(* Schneider Machine Expert - Basic project ProyekAkhir_Izzudin Al Ayyubi_2006574780, file version 2.7.0.0 *)
(* ProjectInformations: Name=New project *)

HARDWARE
  Cpu 0: TM221CE16R
  EthernetConfiguration: NetworkName=M221, IpAllocationMode=FixedAddress, IpAddress=0.0.0.0, SubnetMask=0.0.0.0
  SerialLineConfiguration: Baud=Baud19200, Parity=ParityEven, DataBits=DataBits8, StopBits=StopBits1, PhysicalMedium=PhysicalMediumRs485, TransmissionMode=TransmissionModeModbusRtu, SlaveId=1, Addressing=SlaveAddressing
  MastTask: UsePeriodScanMode=false, PeriodScan=100
  FastTask: Period=255
  CpuBehavior: StartingMode=StartAsPreviousState, AutoSaveRamOnEeprom=true, WatchdogPeriod=250

SYMBOLS  (address, symbol, comment, settings)
  %M0       MOVING_X
  %M2       ITEM_DETECTED
  %M3       LID_AT_PLACE
  %M4       LID_CLAMPED
  %M6       BASE_AT_PLACE
  %M7       BASE_CLAMPED
  %M9       PARTLEAVING
  %M10      START_
  %M11      RESET
  %M12      STOP
  %M13      EMERGENCYS
  %M14      AUTO
  %M16      MACHINE_BUSY
  %M17      RSENSOR1
  %M18      RSENSOR2
  %M19      VS1_1
  %M20      VS1_2
  %M21      VS2_0
  %M22      VS2_1
  %M23      VS2_3
  %M24      MOVE_X
  %M25      MOVE_Z
  %M26      GRAB
  %M27      LIDSCONVEYOR
  %M28      CLAMP_LID
  %M30      BASECONVEYOR
  %M31      CLAMP_BASE
  %M32      POS_RAISE_BASE
  %M33      STARTLIGHT
  %M34      RESETLIGHT
  %M35      STOPLIGHT
  %M36      MACHINE_START
  %M37      MACHINE_STOP
  %M38      MACHINE_RESET
  %M39      CONVEYOR_MC1
  %M40      CONVEYOR_MC2
  %M41      PIVOT_TURN2
  %M42      PIVOT_TURN3
  %M43      PIVOT_BELT2
  %M44      PIVOT_BELT3
  %M45      PRODUCE_LIDS
  %M46      EMITTER
  %M47      BLUELIGHT
  %M100     STARTMEMORY
  %M101     MEMORY2
  %MW0      COUNTER
  %MW1      DIGITALCOUNTER
  %MW2      VSENSOR1
  %MW3      VSENSOR3
  %TM0        [Preset=1, Base=OneSecond]
  %TM1        [Preset=8, Base=OneHundredMilliSeconds]
  %TM2        [Preset=8, Base=OneHundredMilliSeconds]
  %TM3        [Preset=4, Base=OneHundredMilliSeconds]
  %TM4        [Type=TP, Preset=1500, Base=OneHundredMilliSeconds]

POU New POU
  (* SectionNumber=1 *)

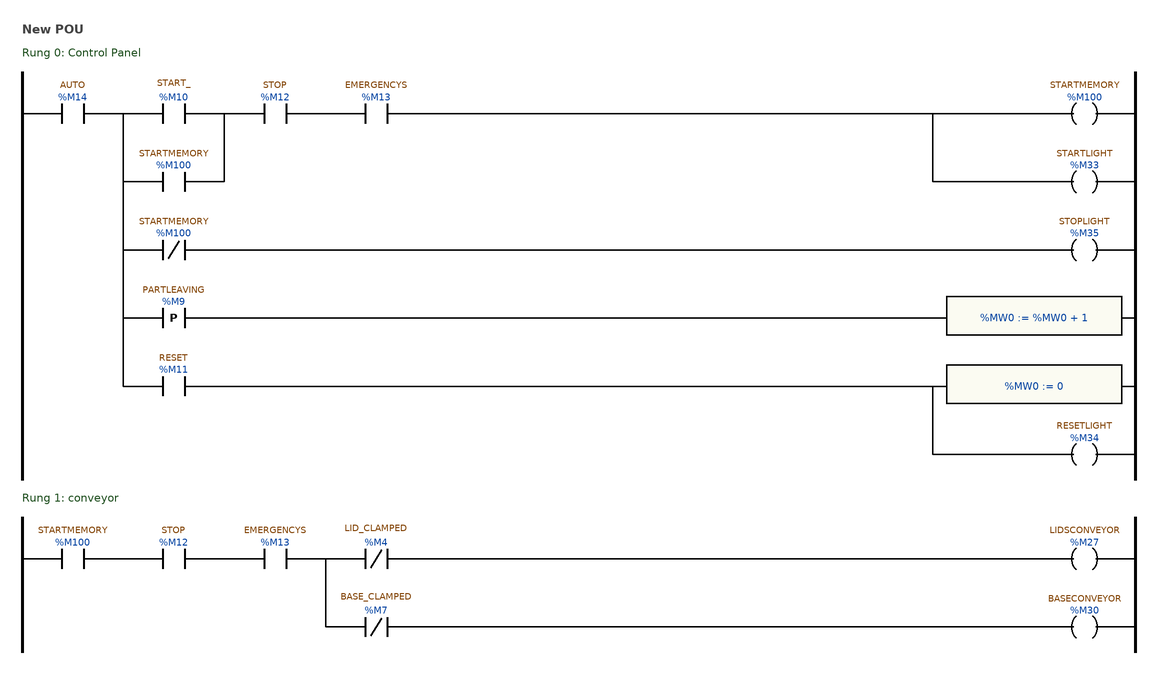

// Rung 0: Control Panel
  LD %M14                 (* AUTO *)
  MPS
  AND( %M10               (* START_ *)
  OR %M100                (* STARTMEMORY *)
  )
  AND %M12                (* STOP *)
  AND %M13                (* EMERGENCYS *)
  ST %M100                (* STARTMEMORY *)
  ST %M33                 (* STARTLIGHT *)
  MRD
  ANDN %M100              (* STARTMEMORY *)
  ST %M35                 (* STOPLIGHT *)
  MRD
  ANDR %M9                (* PARTLEAVING *)
  [ %MW0 := %MW0 + 1 ]    (* COUNTER, COUNTER *)
  MPP
  AND %M11                (* RESET *)
  [ %MW0 := 0 ]           (* COUNTER *)
  ST %M34                 (* RESETLIGHT *)
  // as ST:
  //   _t1 := AUTO AND (START_ OR STARTMEMORY) AND STOP AND EMERGENCYS;
  //   STARTMEMORY := _t1;
  //   STARTLIGHT := _t1;
  //   STOPLIGHT := AUTO AND NOT STARTMEMORY;
  //   IF AUTO AND RISING(PARTLEAVING) THEN COUNTER := COUNTER + 1; END_IF;
  //   IF AUTO AND RESET THEN COUNTER := 0; END_IF;
  //   RESETLIGHT := AUTO AND RESET;

// Rung 1: conveyor
  LD %M100                (* STARTMEMORY *)
  AND %M12                (* STOP *)
  AND %M13                (* EMERGENCYS *)
  MPS
  ANDN %M4                (* LID_CLAMPED *)
  ST %M27                 (* LIDSCONVEYOR *)
  MPP
  ANDN %M7                (* BASE_CLAMPED *)
  ST %M30                 (* BASECONVEYOR *)
  // as ST:
  //   LIDSCONVEYOR := STARTMEMORY AND STOP AND EMERGENCYS AND NOT LID_CLAMPED;
  //   BASECONVEYOR := STARTMEMORY AND STOP AND EMERGENCYS AND NOT BASE_CLAMPED;

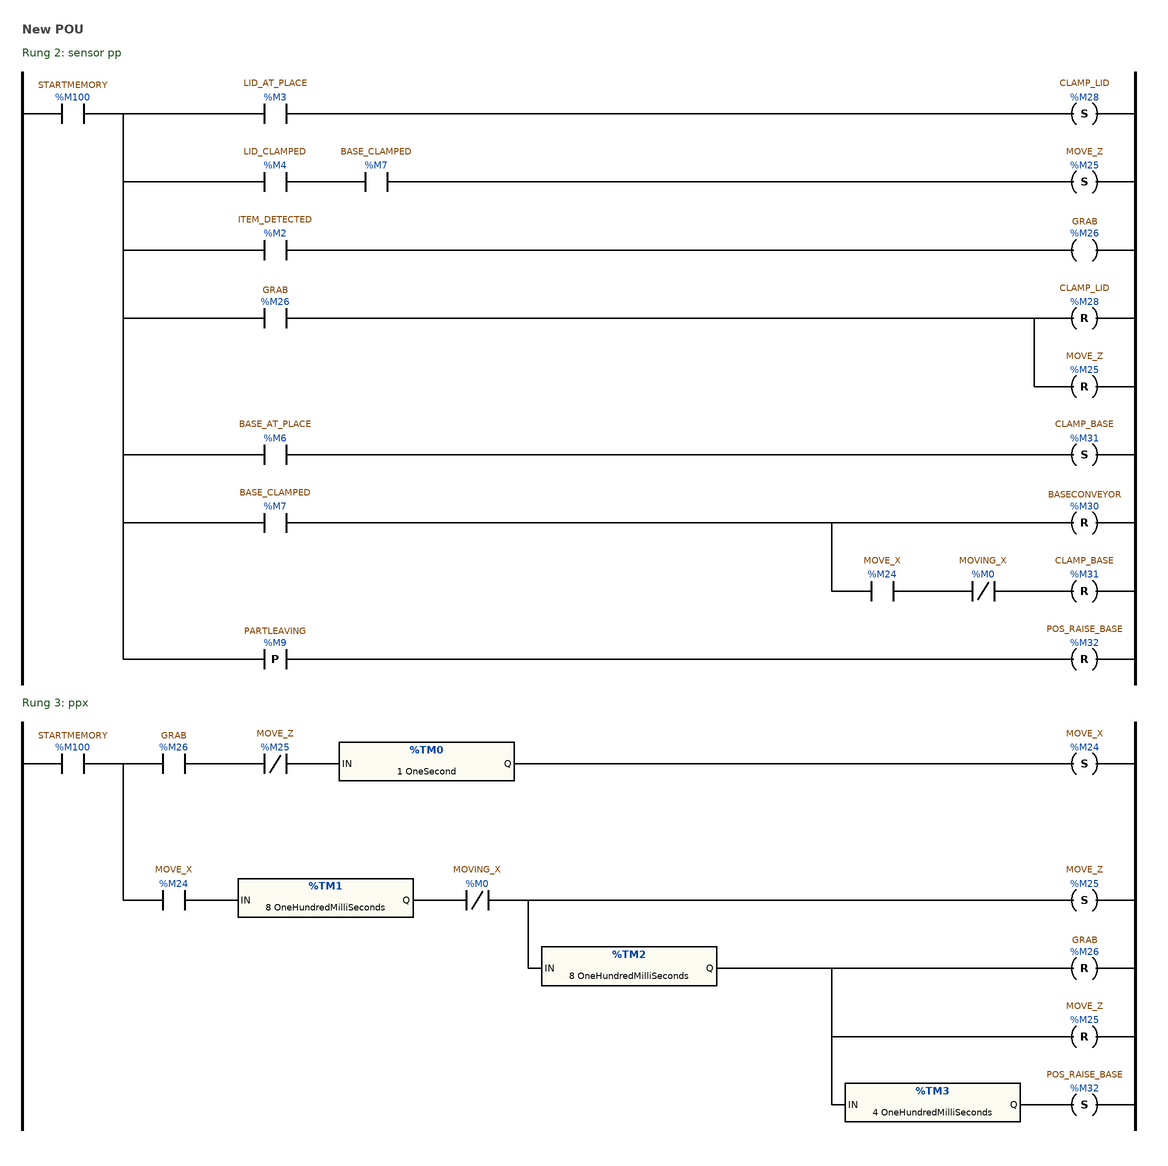

// Rung 2: sensor pp
  LD %M100                (* STARTMEMORY *)
  MPS
  AND %M3                 (* LID_AT_PLACE *)
  S %M28                  (* CLAMP_LID *)
  MRD
  AND %M4                 (* LID_CLAMPED *)
  AND %M7                 (* BASE_CLAMPED *)
  S %M25                  (* MOVE_Z *)
  MRD
  AND %M2                 (* ITEM_DETECTED *)
  ST %M26                 (* GRAB *)
  MRD
  AND %M26                (* GRAB *)
  R %M28                  (* CLAMP_LID *)
  R %M25                  (* MOVE_Z *)
  MRD
  AND %M6                 (* BASE_AT_PLACE *)
  S %M31                  (* CLAMP_BASE *)
  MRD
  AND %M7                 (* BASE_CLAMPED *)
  MPS
  R %M30                  (* BASECONVEYOR *)
  MPP
  AND %M24                (* MOVE_X *)
  ANDN %M0                (* MOVING_X *)
  R %M31                  (* CLAMP_BASE *)
  MPP
  ANDR %M9                (* PARTLEAVING *)
  R %M32                  (* POS_RAISE_BASE *)
  // as ST:
  //   IF STARTMEMORY AND LID_AT_PLACE THEN CLAMP_LID := TRUE; END_IF;
  //   IF STARTMEMORY AND LID_CLAMPED AND BASE_CLAMPED THEN MOVE_Z := TRUE; END_IF;
  //   GRAB := STARTMEMORY AND ITEM_DETECTED;
  //   IF STARTMEMORY AND GRAB THEN CLAMP_LID := FALSE; END_IF;
  //   IF STARTMEMORY AND GRAB THEN MOVE_Z := FALSE; END_IF;
  //   IF STARTMEMORY AND BASE_AT_PLACE THEN CLAMP_BASE := TRUE; END_IF;
  //   IF STARTMEMORY AND BASE_CLAMPED THEN BASECONVEYOR := FALSE; END_IF;
  //   IF STARTMEMORY AND BASE_CLAMPED AND MOVE_X AND NOT MOVING_X THEN CLAMP_BASE := FALSE; END_IF;
  //   IF STARTMEMORY AND RISING(PARTLEAVING) THEN POS_RAISE_BASE := FALSE; END_IF;

// Rung 3: ppx
  LD 1
  MULTIFB
  LD 1
  AND %M100               (* STARTMEMORY *)
  ST %MW2009:X2
  BLK %TM0
  LD %MW2009:X2
  AND %M26                (* GRAB *)
  ANDN %M25               (* MOVE_Z *)
  IN
  OUT_BLK
  LD Q
  S %M24                  (* MOVE_X *)
  END_BLK
  BLK %TM1
  LD %MW2009:X2
  AND %M24                (* MOVE_X *)
  IN
  OUT_BLK
  LD Q
  ST %MW2009:X0
  END_BLK
  LD %MW2009:X0
  ANDN %M0                (* MOVING_X *)
  ST %MW2009:X3
  LD %MW2009:X3
  S %M25                  (* MOVE_Z *)
  BLK %TM2
  LD %MW2009:X3
  IN
  OUT_BLK
  LD Q
  ST %MW2009:X1
  END_BLK
  LD %MW2009:X1
  R %M26                  (* GRAB *)
  R %M25                  (* MOVE_Z *)
  BLK %TM3
  LD %MW2009:X1
  IN
  OUT_BLK
  LD Q
  S %M32                  (* POS_RAISE_BASE *)
  END_BLK
  MULTIFB
  // as ST:
  //   %TM0(IN := STARTMEMORY AND GRAB AND NOT MOVE_Z);
  //   IF %TM0.Q THEN MOVE_X := TRUE; END_IF;
  //   %TM1(IN := STARTMEMORY AND MOVE_X);
  //   IF %TM1.Q AND NOT MOVING_X THEN MOVE_Z := TRUE; END_IF;
  //   %TM2(IN := %TM1.Q AND NOT MOVING_X);
  //   IF %TM2.Q THEN GRAB := FALSE; END_IF;
  //   IF %TM2.Q THEN MOVE_Z := FALSE; END_IF;
  //   %TM3(IN := %TM2.Q);
  //   IF %TM3.Q THEN POS_RAISE_BASE := TRUE; END_IF;

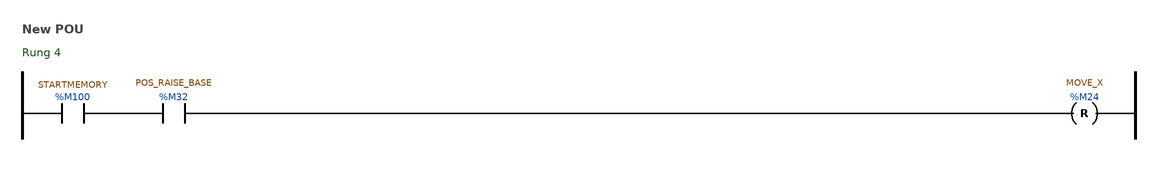

// Rung 4
  LD %M100                (* STARTMEMORY *)
  AND %M32                (* POS_RAISE_BASE *)
  R %M24                  (* MOVE_X *)
  // as ST:
  //   IF STARTMEMORY AND POS_RAISE_BASE THEN MOVE_X := FALSE; END_IF;

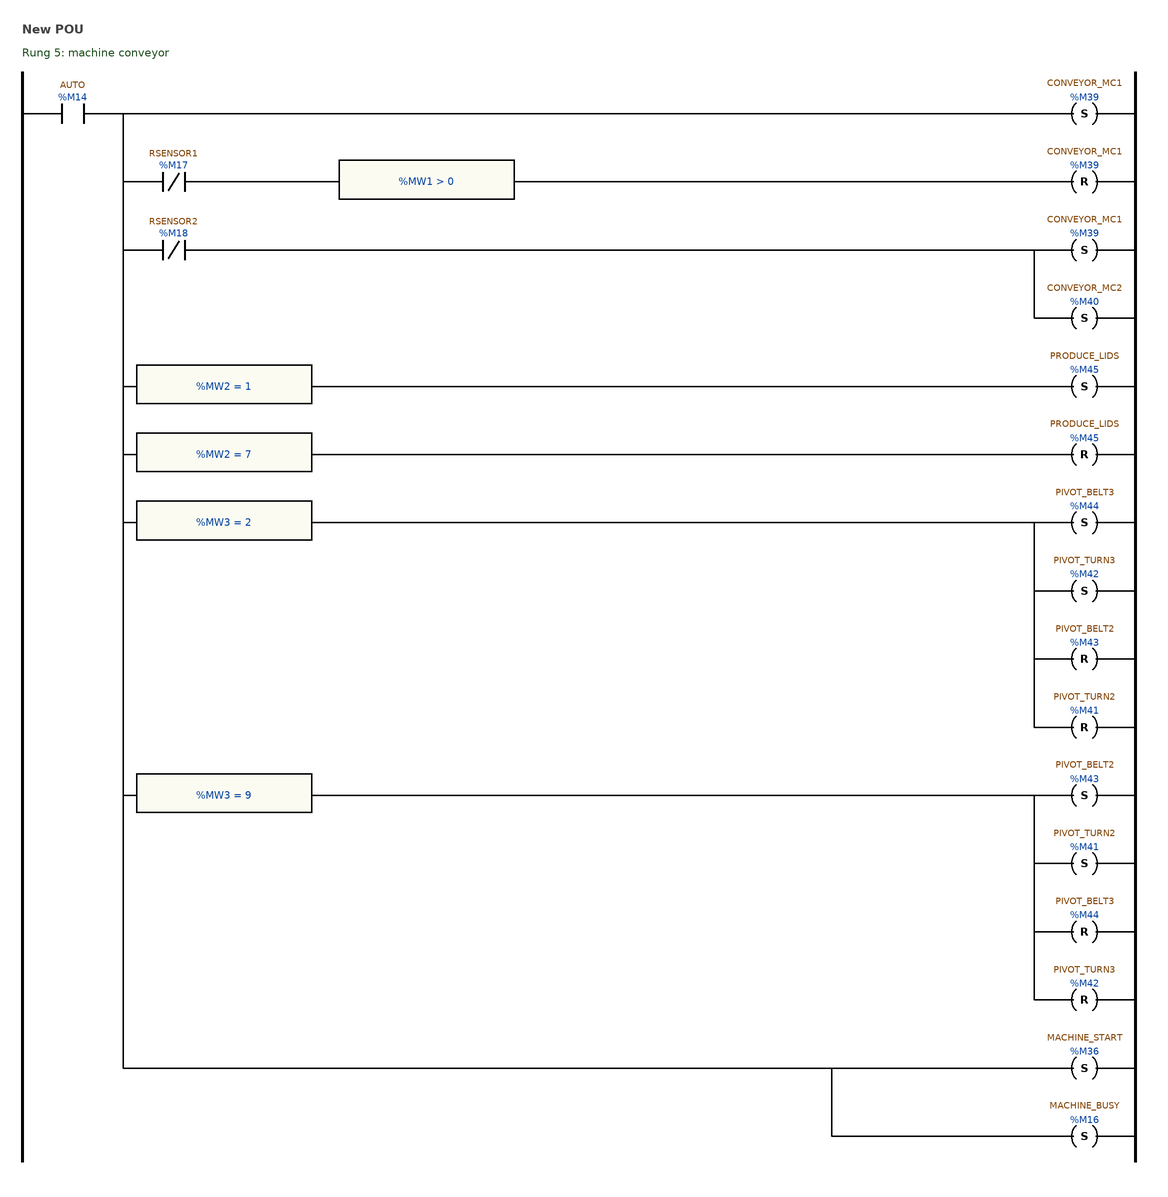

// Rung 5: machine conveyor
  LD %M14                 (* AUTO *)
  MPS
  S %M39                  (* CONVEYOR_MC1 *)
  MRD
  ANDN %M17               (* RSENSOR1 *)
  AND [ %MW1 > 0 ]        (* DIGITALCOUNTER *)
  R %M39                  (* CONVEYOR_MC1 *)
  MRD
  ANDN %M18               (* RSENSOR2 *)
  S %M39                  (* CONVEYOR_MC1 *)
  S %M40                  (* CONVEYOR_MC2 *)
  MRD
  AND [ %MW2 = 1 ]        (* VSENSOR1 *)
  S %M45                  (* PRODUCE_LIDS *)
  MRD
  AND [ %MW2 = 7 ]        (* VSENSOR1 *)
  R %M45                  (* PRODUCE_LIDS *)
  MRD
  AND [ %MW3 = 2 ]        (* VSENSOR3 *)
  S %M44                  (* PIVOT_BELT3 *)
  S %M42                  (* PIVOT_TURN3 *)
  R %M43                  (* PIVOT_BELT2 *)
  R %M41                  (* PIVOT_TURN2 *)
  MRD
  AND [ %MW3 = 9 ]        (* VSENSOR3 *)
  S %M43                  (* PIVOT_BELT2 *)
  S %M41                  (* PIVOT_TURN2 *)
  R %M44                  (* PIVOT_BELT3 *)
  R %M42                  (* PIVOT_TURN3 *)
  MPP
  S %M36                  (* MACHINE_START *)
  S %M16                  (* MACHINE_BUSY *)
  // as ST:
  //   IF AUTO THEN CONVEYOR_MC1 := TRUE; END_IF;
  //   IF AUTO AND NOT RSENSOR1 AND DIGITALCOUNTER > 0 THEN CONVEYOR_MC1 := FALSE; END_IF;
  //   IF AUTO AND NOT RSENSOR2 THEN CONVEYOR_MC1 := TRUE; END_IF;
  //   IF AUTO AND NOT RSENSOR2 THEN CONVEYOR_MC2 := TRUE; END_IF;
  //   IF AUTO AND VSENSOR1 = 1 THEN PRODUCE_LIDS := TRUE; END_IF;
  //   IF AUTO AND VSENSOR1 = 7 THEN PRODUCE_LIDS := FALSE; END_IF;
  //   IF AUTO AND VSENSOR3 = 2 THEN PIVOT_BELT3 := TRUE; END_IF;
  //   IF AUTO AND VSENSOR3 = 2 THEN PIVOT_TURN3 := TRUE; END_IF;
  //   IF AUTO AND VSENSOR3 = 2 THEN PIVOT_BELT2 := FALSE; END_IF;
  //   IF AUTO AND VSENSOR3 = 2 THEN PIVOT_TURN2 := FALSE; END_IF;
  //   IF AUTO AND VSENSOR3 = 9 THEN PIVOT_BELT2 := TRUE; END_IF;
  //   IF AUTO AND VSENSOR3 = 9 THEN PIVOT_TURN2 := TRUE; END_IF;
  //   IF AUTO AND VSENSOR3 = 9 THEN PIVOT_BELT3 := FALSE; END_IF;
  //   IF AUTO AND VSENSOR3 = 9 THEN PIVOT_TURN3 := FALSE; END_IF;
  //   IF AUTO THEN MACHINE_START := TRUE; END_IF;
  //   IF AUTO THEN MACHINE_BUSY := TRUE; END_IF;

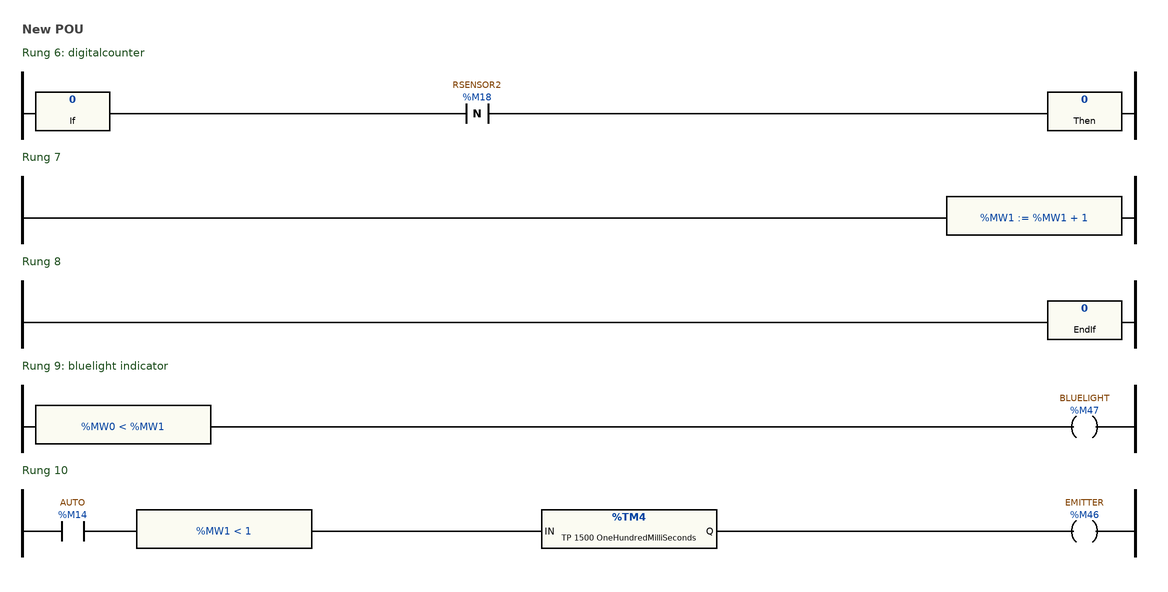

// Rung 6: digitalcounter
  IF0
  ANDF %M18               (* RSENSOR2 *)
  THEN0

// Rung 7
  LD 1
  [ %MW1 := %MW1 + 1 ]    (* DIGITALCOUNTER, DIGITALCOUNTER *)
  // as ST:
  //   DIGITALCOUNTER := DIGITALCOUNTER + 1;

// Rung 8
  LD 1
  ENDIF0

// Rung 9: bluelight indicator
  LD [ %MW0 < %MW1 ]      (* COUNTER, DIGITALCOUNTER *)
  ST %M47                 (* BLUELIGHT *)
  // as ST:
  //   BLUELIGHT := COUNTER < DIGITALCOUNTER;

// Rung 10
  BLK %TM4
  LD %M14                 (* AUTO *)
  AND [ %MW1 < 1 ]        (* DIGITALCOUNTER *)
  IN
  OUT_BLK
  LD Q
  ST %M46                 (* EMITTER *)
  END_BLK
  // as ST:
  //   %TM4(IN := AUTO AND DIGITALCOUNTER < 1);
  //   EMITTER := %TM4.Q;
